{attribute 'qualified_only'}
VAR_GLOBAL
I_LOTBOX_CLAMP_ON_1 AT %I* : BOOL;
I_LOTBOX_CLAMP_ON_2 AT %I* : BOOL;
I_LOTBOX_CLAMP_ON_3 AT %I* : BOOL;
I_LOTBOX_CLAMP_ON_4 AT %I* : BOOL;
I_LOTBOX_CLAMP_OFF_1 AT %I* : BOOL;
I_LOTBOX_CLAMP_OFF_2 AT %I* : BOOL;
I_LOTBOX_CLAMP_OFF_3 AT %I* : BOOL;
I_LOTBOX_CLAMP_OFF_4 AT %I* : BOOL;
	
I_LOTBOX_DETECT_1 AT %I* : BOOL;//LOTBOX_FUKUDA1_DETECT
I_LOTBOX_DETECT_2 AT %I* : BOOL;//LOTBOX_FUKUDA2_DETECT
I_LOTBOX_DETECT_3 AT %I* : BOOL;//LOTBOX_FUKUDA3_DETECT
I_LOTBOX_DETECT_4 AT %I* : BOOL;//LOTBOX_FUKUDA4_DETECT

I_VACUUM_ON AT %I* : BOOL;
I_VACUUM_OFF AT %I* : BOOL;

I_FUKUDA_TRANSFER_AT_FRONT_A AT %I* : BOOL;
I_FUKUDA_TRANSFER_AT_BACK_A AT %I* : BOOL;
I_FUKUDA_TRANSFER_AT_FRONT_B AT %I* : BOOL;
I_FUKUDA_TRANSFER_AT_BACK_B AT %I* : BOOL;
I_FUKUDA_TRANSFER_A_PICK_DONE : BOOL;
I_FUKUDA_TRANSFER_B_PICK_DONE : BOOL;
I_FUKUDA_TRANSFER_AT_A : BOOL;
I_FUKUDA_TRANSFER_AT_B : BOOL;

I_RETURN_DONE_A: BOOL;
I_RETURN_DONE_B: BOOL;
I_LOADING_DONE_A: BOOL;
I_LOADING_DONE_B: BOOL;
I_CURRENT_TRANSACTION : T_CURRENT_TRANSACTION ;
I_FUKUDA_ONDUTY_A:BOOL;
I_FUKUDA_ONDUTY_B:BOOL;
JIG_FUKUDA_PRESENCE: BOOL :=TRUE;

I_LOTEND :BOOL :=TRUE;
I_FUNC_CALLED:BOOL:=TRUE;
I_LOADING_DONE : BOOL;
I_LOADING_FAILED: BOOL;
I_LOADING_ALARM: INT;
I_LOADING_SOCKET : T_JIG_SOCKET;
I_LASER_SOCKET : T_JIG_SOCKET; 
I_CARTESSIAN_GRIPPER_ON AT %I* : BOOL;
I_CARTESSIAN_GRIPPER_OFF AT %I* : BOOL;
I_FUNCTION_NAME :STRING [255];
I_CASE : INT:=0;
I_FUKUDA_RUNNING:BOOL :=FALSE;

O_LOTBOX_CLAMP_ON_1 AT %Q* : BOOL;
O_LOTBOX_CLAMP_ON_2 AT %Q* : BOOL;
O_LOTBOX_CLAMP_ON_3 AT %Q* : BOOL;
O_LOTBOX_CLAMP_ON_4 AT %Q* : BOOL;
O_LOTBOX_CLAMP_OFF_1 AT %Q* : BOOL;
O_LOTBOX_CLAMP_OFF_2 AT %Q* : BOOL;
O_LOTBOX_CLAMP_OFF_3 AT %Q* : BOOL;
O_LOTBOX_CLAMP_OFF_4 AT %Q* : BOOL;

O_VACUUM_ON AT %Q* : BOOL;
O_VACUUM_OFF AT %Q* : BOOL;
O_CARTESSIAN_GRIPPER_ON AT %Q* : BOOL;
O_CARTESSIAN_GRIPPER_OFF AT %Q* : BOOL;
O_TOWER_LAMP_RED AT %Q* : BOOL;
O_TOWER_LAMP_YELLOW AT %Q* : BOOL;
O_TOWER_LAMP_GREEN AT %Q* : BOOL;
O_TOWER_LAMP_BUZZER AT %Q* : BOOL;
O_WARNING_LIGHT AT %Q* : BOOL;
O_LOT_BOX_INDICATOR_1  AT %Q* : BOOL;
O_LOT_BOX_INDICATOR_2 AT %Q* : BOOL;
O_LOT_BOX_INDICATOR_3 AT %Q* : BOOL;
O_LOT_BOX_INDICATOR_4 AT %Q* : BOOL;

AXIS_COMPLETE: BOOL;
LOTBOX_READY_1: BOOL;

DataWordInput1 AT %IB100 : ARRAY [0..15] OF WORD; 
DataWordInput2 AT %IB132 : ARRAY [16..31] OF WORD; 
DataWordInput3 AT %IB164 : ARRAY [32..47] OF WORD; 
DataWordInput4 AT %IB196 : ARRAY [48..56] OF WORD; 
DataWordOutput1 AT %QB100 : ARRAY [0..15] OF WORD; 
DataWordOutput2 AT %QB132 : ARRAY [16..31] OF WORD; 
DataWordOutput3 AT %QB164 : ARRAY [32..47] OF WORD; 
DataWordOutput4 AT %QB196 : ARRAY [48..56] OF WORD; 

I_RETURN_ALARM: INT;
I_RETURN_FAILED: BOOL;
ACTIVE_ID: INT :=1;	
ACTIVE_PROGRAM: INT ;
ACTIVE_PROGRAM_CHANGE:BOOL;
	
I_FUKUDA_HOME : BOOL;
O_FUKUDA_HOME : BOOL; 
STRAIGHTEN_START: BOOL;
STRAIGHTEN_PROCESS: BOOL;
STRAIGHTEN_DONE: BOOL;

FUKUDA_HOME: BOOL;

O_STOPPER_TRANSFER_A AT %Q* : BOOL;
O_STOPPER_TRANSFER_B AT %Q* : BOOL;
I_STOPPER_TRANSFER_ON_A AT %Q* : BOOL;
I_STOPPER_TRANSFER_OFF_A AT %Q* : BOOL;
I_STOPPER_TRANSFER_ON_B AT %Q* : BOOL;
I_STOPPER_TRANSFER_OFF_B AT %Q* : BOOL;
O_RESET_CARTESSIAN AT %Q* : BOOL;

END_VAR

(* stored: Version 1.1.0.1, ProductVersion 3.1.4020.12
   GVL INPUT_VAR: Id {aeaab80c-2fd3-4a23-a84f-fd6d6cc44c78} *)
